Staubli VAL3: getObjectData.pgx

public program getObjectData(num x_nIdx (dimensions=1), num& x_nObjectID[] (dimensions=1), trsf& x_trObject[] (dimensions=1))
begin
  // This program returns the ID number and the coordinates
  // of the detected object.
  //
  // Input param
  // x_nIdx     : Position of the object in the queue
  //
  // Output param
  // x_nObjectID
  // x_trObject   : Coordinates of the object
  //
  // Created 23-02-05                                   C.CURRIVAND
  //----------------------------------------------------------------
  //
  x_nObjectID=nObjectID[x_nIdx]
  x_trObject=trObjectPos[x_nIdx]
end
